{attribute 'pack_mode' := '1'}
TYPE ST_SuspendPathDataIn :
STRUCT
	iPath						: UINT;			// MM path ID (1-65536)
END_STRUCT
END_TYPE

(* stored: Version 1.1.0.1, ProductVersion 3.1.4024.5
   DUT ST_SuspendPathDataIn: Id {837a6b09-e4eb-481e-828f-c28a62af8f26} *)
